// TIA Portal project "indexingStation" (V17)

(* hardware
DEVICE "SCALANCE X005"  SCALANCE X-Station
   slot 0: "Switch_1"  6GK5 005-0BA00-1AB2  V1.0
   slot 0: "SCALANCE X rack"  Rail
DEVICE "ET 200SP station_1"  ET 200SP-Station
   slot 0: "IO device_1"  IM 155-6 PN/2 HF  6ES7 155-6AU01-0CN0  V4.2
   slot 0: "Rack_0"  Rack  6ES5 710-8MAx1
   slot 1: "DI 8x24VDC HF_1"  DI 8x24VDC HF  6ES7 131-6BF00-0CA0  V2.0
      slot 1: "DI 8x24VDC HF_1"  DI 8x24VDC HF
   slot 2: "DI 8x24VDC HF_2"  DI 8x24VDC HF  6ES7 131-6BF00-0CA0  V2.0
      slot 1: "DI 8x24VDC HF_2"  DI 8x24VDC HF
   slot 3: "DI 8x24VDC HF_3"  DI 8x24VDC HF  6ES7 131-6BF00-0CA0  V2.0
      slot 1: "DI 8x24VDC HF_3"  DI 8x24VDC HF
   slot 4: "DQ 8x24VDC/0.5A HF_1"  DQ 8x24VDC/0.5A HF  6ES7 132-6BF00-0CA0  V2.0
      slot 1: "DQ 8x24VDC/0.5A HF_1"  DQ 8x24VDC/0.5A HF
   slot 5: "DQ 8x24VDC/0.5A HF_2"  DQ 8x24VDC/0.5A HF  6ES7 132-6BF00-0CA0  V2.0
      slot 1: "DQ 8x24VDC/0.5A HF_2"  DQ 8x24VDC/0.5A HF
   slot 6: "Server module_1"  Server module  6ES7 193-6PA00-0AA0  V1.1
      slot 1: "Server module_1"  Server module
   slot 127: "BA 2xRJ45"  BA 2xRJ45  6ES7 193-6AR00-0AA0  V0.0
      slot 1: "Port_1"  X1 P1 R  6ES7 193-6AR00-0AA0  V0.0
      slot 2: "Port_2"  X1 P2 R  6ES7 193-6AR00-0AA0  V0.0
DEVICE "S7-1200 station_1"  S7-1200 Station
   slot 0: "Rack_0"  S7-1200 Rack  Rack  V1.0
   slot 1: "PLC_1"  CPU 1214C DC/DC/DC  6ES7 214-1AG40-0XB0  V4.4
*)

// ===== PLC "PLC_1"  CPU 1214C DC/DC/DC =====

VAR_GLOBAL   // PLC tag table "Default tag table"
   "wrong orientation" AT %M10.0 : Bool;
   "Tag_1" AT %M202.1 : Bool;
   "end check" AT %M10.1 : Bool;
   "start correction" AT %M10.2 : Bool;
   "Tag_2" AT %M202.2 : Bool;
   "initiateGripper" AT %M10.3 : Bool;
   "initiateLifting" AT %M10.4 : Bool;
   "initiateRotation" AT %M10.5 : Bool;
   "initiateReturn" AT %M10.6 : Bool;
   "Tag_3" AT %M202.3 : Bool;
   "initiateOpenGripper" AT %M10.7 : Bool;
   "initiateNormalcy" AT %M11.0 : Bool;
   "Tag_4" AT %M202.4 : Bool;
   "initiateStepperMotor" AT %M11.1 : Bool;
   "prepForTransfer" AT %M11.2 : Bool;
   "initiateRetractionAfterTransfer" AT %M11.3 : Bool;
   "Clock_Byte" AT %MB50 : Byte;
   "Clock_10Hz" AT %M50.0 : Bool;
   "Clock_5Hz" AT %M50.1 : Bool;
   "Clock_2.5Hz" AT %M50.2 : Bool;
   "Clock_2Hz" AT %M50.3 : Bool;
   "Clock_1.25Hz" AT %M50.4 : Bool;
   "Clock_1Hz" AT %M50.5 : Bool;
   "Clock_0.625Hz" AT %M50.6 : Bool;
   "Clock_0.5Hz" AT %M50.7 : Bool;
   "rotate for check" AT %M11.4 : Bool;
   "rotate 90 if correct" AT %M11.5 : Bool;
   "rotate 45 if correct" AT %M11.6 : Bool;
   "rotate45 if incorrect" AT %M11.7 : Bool;
   "rotate 90 after incorrect orientation" AT %M12.0 : Bool;
END_VAR

VAR_GLOBAL   // PLC tag table "OurInputsAndOutputs"
   "Auto switch" AT %I0.6 : Bool;
   "reset Switch" AT %I0.5 : Bool;
   "start button" AT %I2.3 : Bool;
   "stop button" AT %I2.4 : Bool;
   "emergency stop" AT %I2.5 : Bool;
   "output power on" AT %I2.6 : Bool;
   "input 1 from previous station" AT %I2.7 : Bool;
   "input 2 from previous station" AT %I3.0 : Bool;
   "input 1 from next station" AT %I3.1 : Bool;
   "input 2 from next station" AT %I3.2 : Bool;
   "transfer cylinder 4A retracted" AT %I3.3 : Bool;
   "transfer cylinder 4A extended" AT %I3.4 : Bool;
   "lift cylinder 1A retracted" AT %I3.5 : Bool;
   "lift cylinder 1A extended" AT %I3.6 : Bool;
   "port present(orientationposition)" AT %I3.7 : Bool;
   "rotation cylinder 2A retracted" AT %I4.0 : Bool;
   "rotation cylinder 2A extended" AT %I4.1 : Bool;
   "Spool upper port detected" AT %I4.2 : Bool;
   "indexing station in home position" AT %I4.3 : Bool;
   "stepper motor ready" AT %I4.4 : Bool;
   "part present(initial position)" AT %I4.5 : Bool;
   "automatic on(green)" AT %Q2.0 : Bool;
   "output 1 to previous station" AT %Q2.1 : Bool;
   "output 2 to previous station" AT %Q2.2 : Bool;
   "output 1 to next station" AT %Q2.3 : Bool;
   "output 2 to next station" AT %Q2.4 : Bool;
   "extend transfer cylinder 3A" AT %Q2.5 : Bool;
   "extend lift cylinder" AT %Q2.6 : Bool;
   "retract lift cylinder" AT %Q2.7 : Bool;
   "stepper motor M1 go 45" AT %Q3.2 : Bool;
   "stepper motor M1 go 90" AT %Q3.3 : Bool;
   "release gripper 3A" AT %Q3.4 : Bool;
   "close gripper 3A" AT %Q3.5 : Bool;
   "extend rotation cylinder" AT %Q3.6 : Bool;
   "retract rotatioin cylinder" AT %Q3.7 : Bool;
END_VAR

// folder: System blocks/Program resources

DATA_BLOCK "timer 1"   // DB1
{ S7_Optimized_Access := 'TRUE' }
AUTHOR : Simatic
FAMILY : IEC
NAME : IEC_TMR
VERSION : 1.0
// stored: InstanceOfName IEC_TIMER
"IEC_TIMER"
BEGIN
END_DATA_BLOCK

DATA_BLOCK "timer 2"   // DB3
{ S7_Optimized_Access := 'TRUE' }
AUTHOR : Simatic
FAMILY : IEC
NAME : IEC_TMR
VERSION : 1.0
// stored: InstanceOfName IEC_TIMER
"IEC_TIMER"
BEGIN
END_DATA_BLOCK

DATA_BLOCK "timer 3"   // DB4
{ S7_Optimized_Access := 'TRUE' }
AUTHOR : Simatic
FAMILY : IEC
NAME : IEC_TMR
VERSION : 1.0
// stored: InstanceOfName IEC_TIMER
"IEC_TIMER"
BEGIN
END_DATA_BLOCK

DATA_BLOCK "timer 4"   // DB5
{ S7_Optimized_Access := 'TRUE' }
AUTHOR : Simatic
FAMILY : IEC
NAME : IEC_TMR
VERSION : 1.0
// stored: InstanceOfName IEC_TIMER
"IEC_TIMER"
BEGIN
END_DATA_BLOCK

// folder: (top level)

FUNCTION "correct orientation" : Void   // FC1, LAD
{ S7_Optimized_Access := 'TRUE' }
VERSION : 0.1
BEGIN

REGION Network 1: moving the stepper motor by 135 degrees
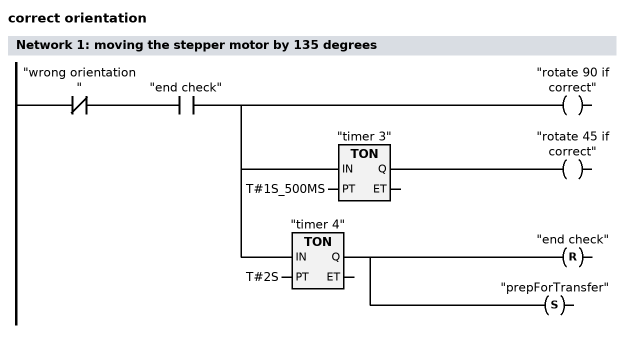
   "rotate 90 if correct" := NOT "wrong orientation" AND "end check";
   "timer 3".TON(IN := "rotate 90 if correct", PT := T#1S_500MS);
   "rotate 45 if correct" := "timer 3".Q;
   "timer 4".TON(IN := "rotate 90 if correct", PT := T#2S);
   IF "timer 4".Q THEN
       "end check" := FALSE;
       "prepForTransfer" := TRUE;
   END_IF;
END_REGION
END_FUNCTION

FUNCTION "incorrect orientation" : Void   // FC2, LAD
{ S7_Optimized_Access := 'TRUE' }
VERSION : 0.1
   VAR_TEMP   // added for the SCL form of the ladder/FBD networks
      _w1 : Bool;
   END_VAR
BEGIN

REGION Network 1: Launching of the correction procedure
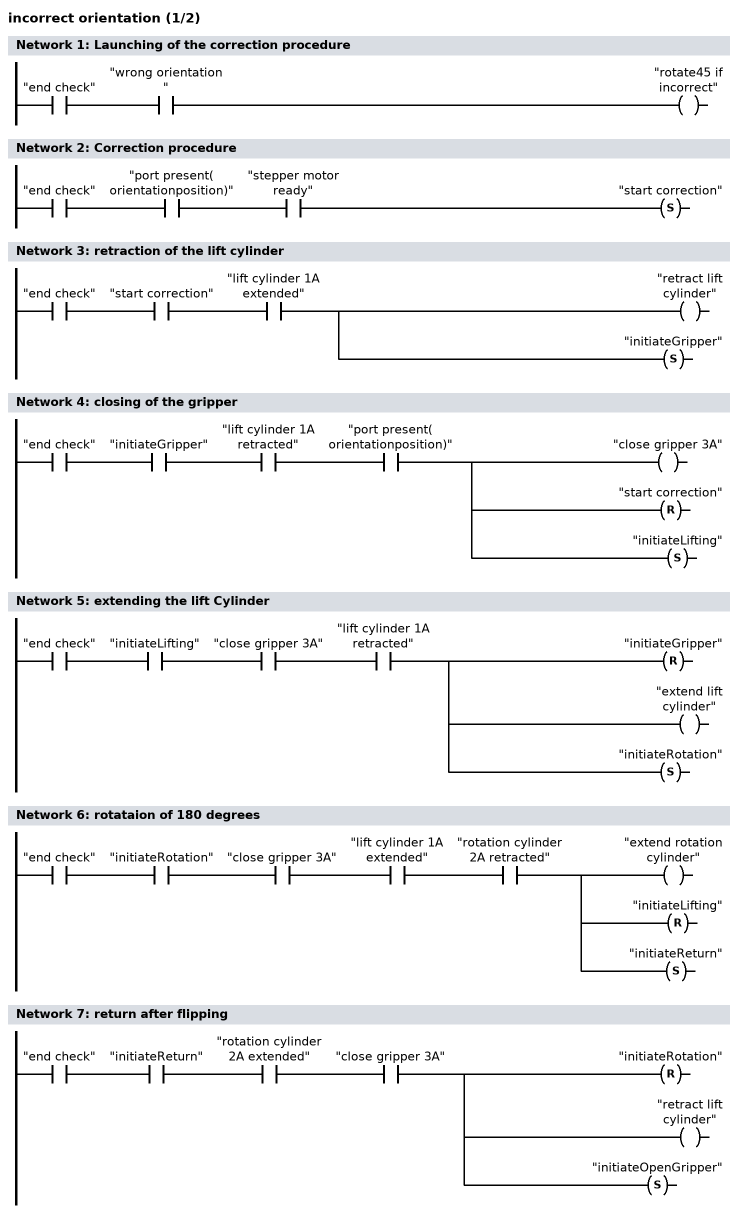
   RUNG wire#powerrail
      Contact( "end check" )
      Contact( "wrong orientation" )
      Coil( "rotate45 if incorrect" )
   END_RUNG
   // the same network as SCL:
   "rotate45 if incorrect" := "end check" AND "wrong orientation";
END_REGION

REGION Network 2: Correction procedure
   RUNG wire#powerrail
      Contact( "end check" )
      Contact( "port present(orientationposition)" )
      Contact( "stepper motor ready" )
      S_Coil( "start correction" )
   END_RUNG
   // the same network as SCL:
   IF "end check" AND "port present(orientationposition)" AND "stepper motor ready" THEN
       "start correction" := TRUE;
   END_IF;
END_REGION

REGION Network 3: retraction of the lift cylinder
   RUNG wire#powerrail
      Contact( "end check" )
      Contact( "start correction" )
      Contact( "lift cylinder 1A extended" )
      wire#w1
      Coil( "retract lift cylinder" )
   END_RUNG
   RUNG wire#w1
      S_Coil( "initiateGripper" )
   END_RUNG
   // the same network as SCL:
   "retract lift cylinder" := "end check" AND "start correction" AND "lift cylinder 1A extended";
   IF "retract lift cylinder" THEN "initiateGripper" := TRUE; END_IF;
END_REGION

REGION Network 4: closing of the gripper
   RUNG wire#powerrail
      Contact( "end check" )
      Contact( "initiateGripper" )
      Contact( "lift cylinder 1A retracted" )
      Contact( "port present(orientationposition)" )
      wire#w1
      Coil( "close gripper 3A" )
   END_RUNG
   RUNG wire#w1
      R_Coil( "start correction" )
   END_RUNG
   RUNG wire#w1
      S_Coil( "initiateLifting" )
   END_RUNG
   // the same network as SCL:
   "close gripper 3A" := "end check" AND "initiateGripper" AND "lift cylinder 1A retracted" AND "port present(orientationposition)";
   IF "close gripper 3A" THEN
       "start correction" := FALSE;
       "initiateLifting" := TRUE;
   END_IF;
END_REGION

REGION Network 5: extending the lift Cylinder
   RUNG wire#powerrail
      Contact( "end check" )
      Contact( "initiateLifting" )
      Contact( "close gripper 3A" )
      Contact( "lift cylinder 1A retracted" )
      wire#w1
      R_Coil( "initiateGripper" )
   END_RUNG
   RUNG wire#w1
      Coil( "extend lift cylinder" )
   END_RUNG
   RUNG wire#w1
      S_Coil( "initiateRotation" )
   END_RUNG
   // the same network as SCL:
   #_w1 := "end check" AND "initiateLifting" AND "close gripper 3A" AND "lift cylinder 1A retracted";
   IF #_w1 THEN "initiateGripper" := FALSE; END_IF;
   "extend lift cylinder" := #_w1;
   IF #_w1 THEN "initiateRotation" := TRUE; END_IF;
END_REGION

REGION Network 6: rotataion of 180 degrees
   RUNG wire#powerrail
      Contact( "end check" )
      Contact( "initiateRotation" )
      Contact( "close gripper 3A" )
      Contact( "lift cylinder 1A extended" )
      Contact( "rotation cylinder 2A retracted" )
      wire#w1
      Coil( "extend rotation cylinder" )
   END_RUNG
   RUNG wire#w1
      R_Coil( "initiateLifting" )
   END_RUNG
   RUNG wire#w1
      S_Coil( "initiateReturn" )
   END_RUNG
   // the same network as SCL:
   "extend rotation cylinder" := "end check" AND "initiateRotation" AND "close gripper 3A" AND "lift cylinder 1A extended" AND "rotation cylinder 2A retracted";
   IF "extend rotation cylinder" THEN
       "initiateLifting" := FALSE;
       "initiateReturn" := TRUE;
   END_IF;
END_REGION

REGION Network 7: return after flipping
   RUNG wire#powerrail
      Contact( "end check" )
      Contact( "initiateReturn" )
      Contact( "rotation cylinder 2A extended" )
      Contact( "close gripper 3A" )
      wire#w1
      R_Coil( "initiateRotation" )
   END_RUNG
   RUNG wire#w1
      Coil( "retract lift cylinder" )
   END_RUNG
   RUNG wire#w1
      S_Coil( "initiateOpenGripper" )
   END_RUNG
   // the same network as SCL:
   #_w1 := "end check" AND "initiateReturn" AND "rotation cylinder 2A extended" AND "close gripper 3A";
   IF #_w1 THEN "initiateRotation" := FALSE; END_IF;
   "retract lift cylinder" := #_w1;
   IF #_w1 THEN "initiateOpenGripper" := TRUE; END_IF;
END_REGION

REGION Network 8: releasing gripper
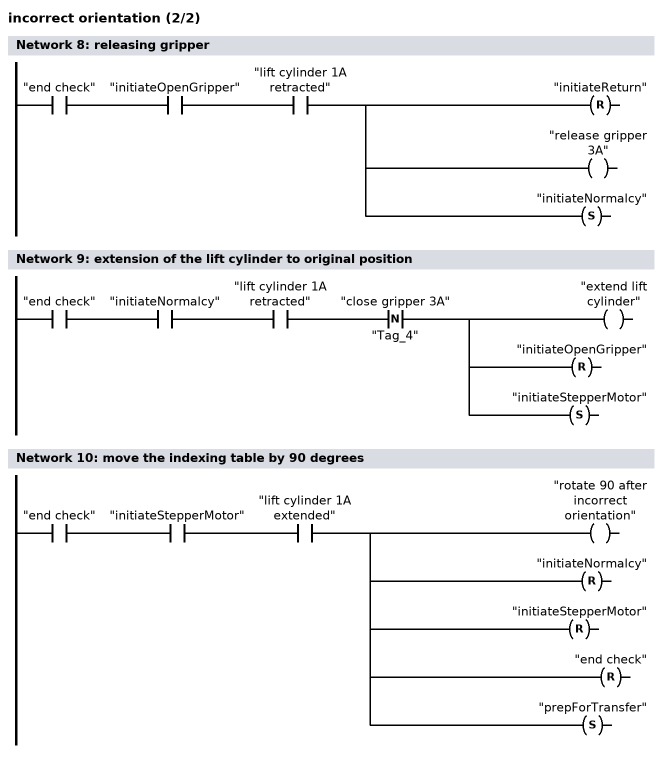
   RUNG wire#powerrail
      Contact( "end check" )
      Contact( "initiateOpenGripper" )
      Contact( "lift cylinder 1A retracted" )
      wire#w1
      R_Coil( "initiateReturn" )
   END_RUNG
   RUNG wire#w1
      Coil( "release gripper 3A" )
   END_RUNG
   RUNG wire#w1
      S_Coil( "initiateNormalcy" )
   END_RUNG
   // the same network as SCL:
   #_w1 := "end check" AND "initiateOpenGripper" AND "lift cylinder 1A retracted";
   IF #_w1 THEN "initiateReturn" := FALSE; END_IF;
   "release gripper 3A" := #_w1;
   IF #_w1 THEN "initiateNormalcy" := TRUE; END_IF;
END_REGION

REGION Network 9: extension of the lift cylinder to original position
   RUNG wire#powerrail
      Contact( "end check" )
      Contact( "initiateNormalcy" )
      Contact( "lift cylinder 1A retracted" )
      N_Contact(operand := "close gripper 3A", bit := "Tag_4")
      wire#w1
      Coil( "extend lift cylinder" )
   END_RUNG
   RUNG wire#w1
      R_Coil( "initiateOpenGripper" )
   END_RUNG
   RUNG wire#w1
      S_Coil( "initiateStepperMotor" )
   END_RUNG
   // the same network as SCL:
   #_w1 := "end check" AND "initiateNormalcy" AND "lift cylinder 1A retracted" AND NOT "close gripper 3A" AND "Tag_4";   // falling edge of "close gripper 3A"
   "Tag_4" := "close gripper 3A";
   "extend lift cylinder" := #_w1;
   IF #_w1 THEN
       "initiateOpenGripper" := FALSE;
       "initiateStepperMotor" := TRUE;
   END_IF;
END_REGION

REGION Network 10: move the indexing table by 90 degrees
   RUNG wire#powerrail
      Contact( "end check" )
      Contact( "initiateStepperMotor" )
      Contact( "lift cylinder 1A extended" )
      wire#w1
      Coil( "rotate 90 after incorrect orientation" )
   END_RUNG
   RUNG wire#w1
      R_Coil( "initiateNormalcy" )
   END_RUNG
   RUNG wire#w1
      R_Coil( "initiateStepperMotor" )
   END_RUNG
   RUNG wire#w1
      R_Coil( "end check" )
   END_RUNG
   RUNG wire#w1
      S_Coil( "prepForTransfer" )
   END_RUNG
   // the same network as SCL:
   "rotate 90 after incorrect orientation" := "end check" AND "initiateStepperMotor" AND "lift cylinder 1A extended";
   IF "rotate 90 after incorrect orientation" THEN
       "initiateNormalcy" := FALSE;
       "initiateStepperMotor" := FALSE;
       "end check" := FALSE;
       "prepForTransfer" := TRUE;
   END_IF;
END_REGION
END_FUNCTION

FUNCTION "Block_1" : Void   // FC3, LAD
{ S7_Optimized_Access := 'TRUE' }
VERSION : 0.1
BEGIN

REGION Network 1
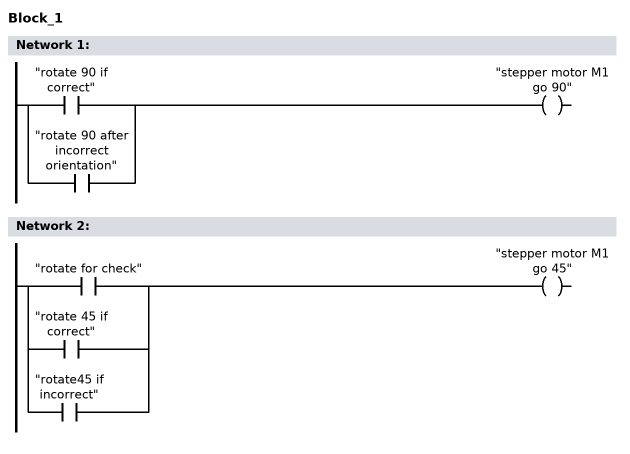
   RUNG wire#powerrail
      Contact( "rotate 90 if correct" )
      wire#w1
      Coil( "stepper motor M1 go 90" )
   END_RUNG
   RUNG wire#powerrail
      Contact( "rotate 90 after incorrect orientation" )
   END_RUNG wire#w1
   // the same network as SCL:
   "stepper motor M1 go 90" := "rotate 90 if correct" OR "rotate 90 after incorrect orientation";
END_REGION

REGION Network 2
   RUNG wire#powerrail
      Contact( "rotate for check" )
      wire#w1
      Coil( "stepper motor M1 go 45" )
   END_RUNG
   RUNG wire#powerrail
      Contact( "rotate 45 if correct" )
   END_RUNG wire#w1
   RUNG wire#powerrail
      Contact( "rotate45 if incorrect" )
   END_RUNG wire#w1
   // the same network as SCL:
   "stepper motor M1 go 45" := "rotate for check" OR "rotate 45 if correct" OR "rotate45 if incorrect";
END_REGION
END_FUNCTION

ORGANIZATION_BLOCK "Main"   // OB1, LAD, ProgramCycle
TITLE = "Main Program Sweep (Cycle)"
{ S7_Optimized_Access := 'TRUE' }
VERSION : 0.1
   VAR_INPUT
      Initial_Call : Bool;   // Initial call of this OB
      Remanence : Bool;   // =True, if remanent data are available
   END_VAR
   VAR_TEMP   // added for the SCL form of the ladder/FBD networks
      _w1 : Bool;
   END_VAR
BEGIN

REGION Network 1: Stepper motor go 45
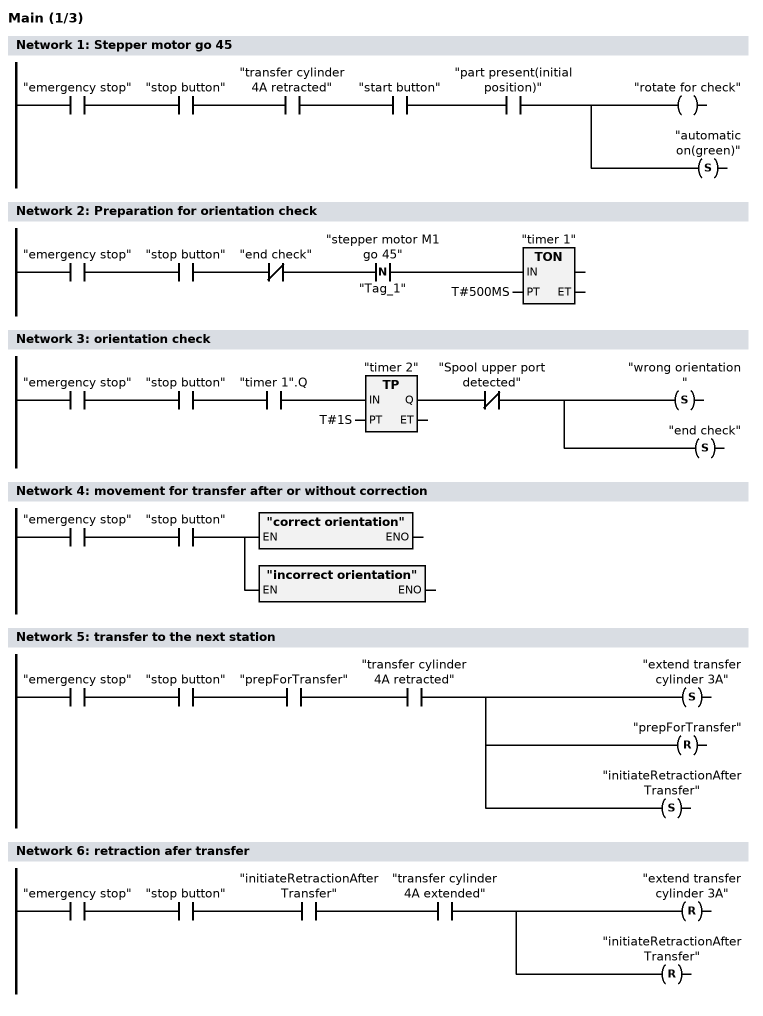
   RUNG wire#powerrail
      Contact( "emergency stop" )
      Contact( "stop button" )
      Contact( "transfer cylinder 4A retracted" )
      Contact( "start button" )
      Contact( "part present(initial position)" )
      wire#w1
      Coil( "rotate for check" )
   END_RUNG
   RUNG wire#w1
      S_Coil( "automatic on(green)" )
   END_RUNG
   // the same network as SCL:
   "rotate for check" := "emergency stop" AND "stop button" AND "transfer cylinder 4A retracted" AND "start button" AND "part present(initial position)";
   IF "rotate for check" THEN "automatic on(green)" := TRUE; END_IF;
END_REGION

REGION Network 2: Preparation for orientation check
   #_w1 := "emergency stop" AND "stop button" AND NOT "end check" AND NOT "stepper motor M1 go 45" AND "Tag_1";   // falling edge of "stepper motor M1 go 45"
   "Tag_1" := "stepper motor M1 go 45";
   "timer 1".TON(IN := #_w1, PT := T#500MS);
END_REGION

REGION Network 3: orientation check
   "timer 2".TP(IN := "emergency stop" AND "stop button" AND "timer 1".Q, PT := T#1S);
   IF "timer 2".Q AND NOT "Spool upper port detected" THEN
       "wrong orientation" := TRUE;
       "end check" := TRUE;
   END_IF;
END_REGION

REGION Network 4: movement for transfer after or without correction
   RUNG wire#powerrail
      Contact( "emergency stop" )
      Contact( "stop button" )
      wire#w1
      "correct orientation"()
   END_RUNG
   RUNG wire#w1
      "incorrect orientation"()
   END_RUNG
   // the same network as SCL:
   #_w1 := "emergency stop" AND "stop button";
   IF #_w1 THEN
       "correct orientation"();
       "incorrect orientation"();
   END_IF;
END_REGION

REGION Network 5: transfer to the next station
   RUNG wire#powerrail
      Contact( "emergency stop" )
      Contact( "stop button" )
      Contact( "prepForTransfer" )
      Contact( "transfer cylinder 4A retracted" )
      wire#w1
      S_Coil( "extend transfer cylinder 3A" )
   END_RUNG
   RUNG wire#w1
      R_Coil( "prepForTransfer" )
   END_RUNG
   RUNG wire#w1
      S_Coil( "initiateRetractionAfterTransfer" )
   END_RUNG
   // the same network as SCL:
   IF "emergency stop" AND "stop button" AND "prepForTransfer" AND "transfer cylinder 4A retracted" THEN
       "extend transfer cylinder 3A" := TRUE;
   END_IF;
   #_w1 := "emergency stop" AND "stop button" AND "prepForTransfer" AND "transfer cylinder 4A retracted";
   IF #_w1 THEN
       "prepForTransfer" := FALSE;
       "initiateRetractionAfterTransfer" := TRUE;
   END_IF;
END_REGION

REGION Network 6: retraction afer transfer
   RUNG wire#powerrail
      Contact( "emergency stop" )
      Contact( "stop button" )
      Contact( "initiateRetractionAfterTransfer" )
      Contact( "transfer cylinder 4A extended" )
      wire#w1
      R_Coil( "extend transfer cylinder 3A" )
   END_RUNG
   RUNG wire#w1
      R_Coil( "initiateRetractionAfterTransfer" )
   END_RUNG
   // the same network as SCL:
   IF "emergency stop" AND "stop button" AND "initiateRetractionAfterTransfer" AND "transfer cylinder 4A extended" THEN
       "extend transfer cylinder 3A" := FALSE;
       "initiateRetractionAfterTransfer" := FALSE;
   END_IF;
END_REGION

REGION Network 7: reset action
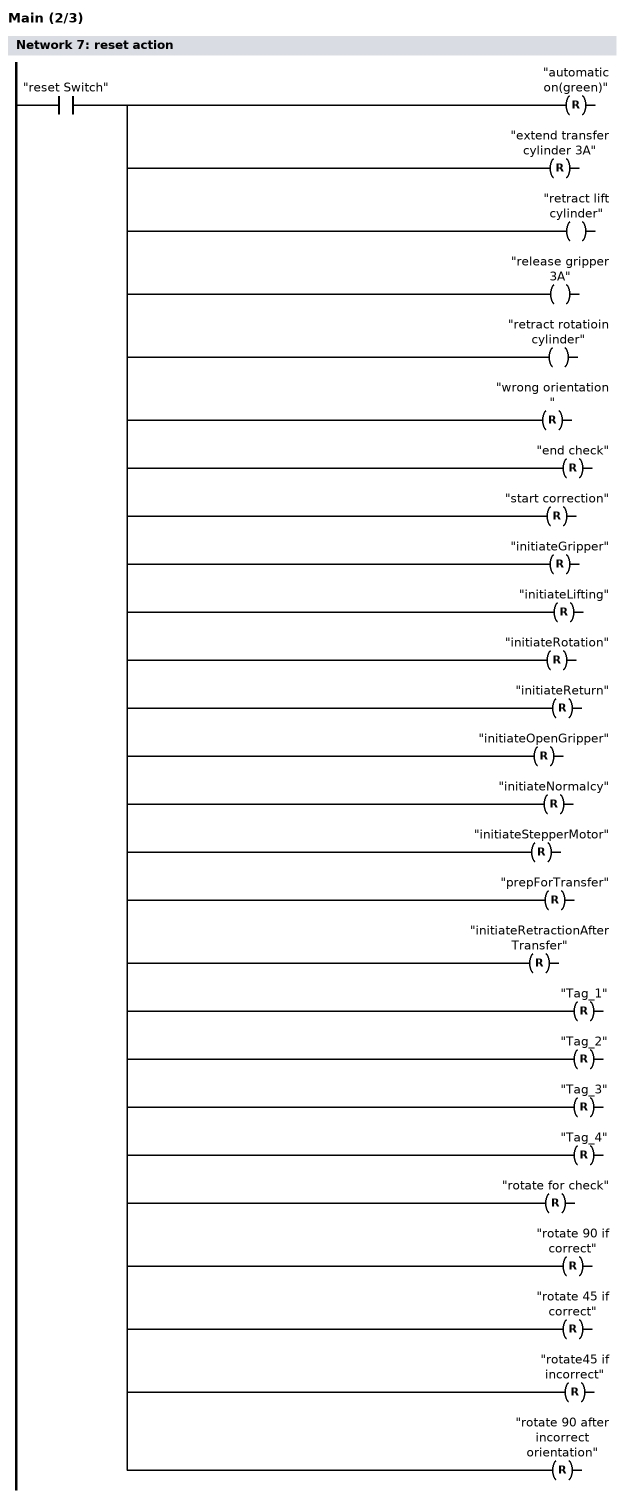
   RUNG wire#powerrail
      Contact( "reset Switch" )
      wire#w1
      R_Coil( "automatic on(green)" )
   END_RUNG
   RUNG wire#w1
      R_Coil( "extend transfer cylinder 3A" )
   END_RUNG
   RUNG wire#w1
      Coil( "retract lift cylinder" )
   END_RUNG
   RUNG wire#w1
      Coil( "release gripper 3A" )
   END_RUNG
   RUNG wire#w1
      Coil( "retract rotatioin cylinder" )
   END_RUNG
   RUNG wire#w1
      R_Coil( "wrong orientation" )
   END_RUNG
   RUNG wire#w1
      R_Coil( "end check" )
   END_RUNG
   RUNG wire#w1
      R_Coil( "start correction" )
   END_RUNG
   RUNG wire#w1
      R_Coil( "initiateGripper" )
   END_RUNG
   RUNG wire#w1
      R_Coil( "initiateLifting" )
   END_RUNG
   RUNG wire#w1
      R_Coil( "initiateRotation" )
   END_RUNG
   RUNG wire#w1
      R_Coil( "initiateReturn" )
   END_RUNG
   RUNG wire#w1
      R_Coil( "initiateOpenGripper" )
   END_RUNG
   RUNG wire#w1
      R_Coil( "initiateNormalcy" )
   END_RUNG
   RUNG wire#w1
      R_Coil( "initiateStepperMotor" )
   END_RUNG
   RUNG wire#w1
      R_Coil( "prepForTransfer" )
   END_RUNG
   RUNG wire#w1
      R_Coil( "initiateRetractionAfterTransfer" )
   END_RUNG
   RUNG wire#w1
      R_Coil( "Tag_1" )
   END_RUNG
   RUNG wire#w1
      R_Coil( "Tag_2" )
   END_RUNG
   RUNG wire#w1
      R_Coil( "Tag_3" )
   END_RUNG
   RUNG wire#w1
      R_Coil( "Tag_4" )
   END_RUNG
   RUNG wire#w1
      R_Coil( "rotate for check" )
   END_RUNG
   RUNG wire#w1
      R_Coil( "rotate 90 if correct" )
   END_RUNG
   RUNG wire#w1
      R_Coil( "rotate 45 if correct" )
   END_RUNG
   RUNG wire#w1
      R_Coil( "rotate45 if incorrect" )
   END_RUNG
   RUNG wire#w1
      R_Coil( "rotate 90 after incorrect orientation" )
   END_RUNG
   // the same network as SCL:
   IF "reset Switch" THEN
       "automatic on(green)" := FALSE;
       "extend transfer cylinder 3A" := FALSE;
   END_IF;
   "retract lift cylinder" := "reset Switch";
   "release gripper 3A" := "reset Switch";
   "retract rotatioin cylinder" := "reset Switch";
   IF "reset Switch" THEN
       "wrong orientation" := FALSE;
       "end check" := FALSE;
       "start correction" := FALSE;
       "initiateGripper" := FALSE;
       "initiateLifting" := FALSE;
       "initiateRotation" := FALSE;
       "initiateReturn" := FALSE;
       "initiateOpenGripper" := FALSE;
       "initiateNormalcy" := FALSE;
       "initiateStepperMotor" := FALSE;
       "prepForTransfer" := FALSE;
       "initiateRetractionAfterTransfer" := FALSE;
       "Tag_1" := FALSE;
       "Tag_2" := FALSE;
       "Tag_3" := FALSE;
       "Tag_4" := FALSE;
       "rotate for check" := FALSE;
       "rotate 90 if correct" := FALSE;
       "rotate 45 if correct" := FALSE;
       "rotate45 if incorrect" := FALSE;
       "rotate 90 after incorrect orientation" := FALSE;
   END_IF;
END_REGION

REGION Network 8
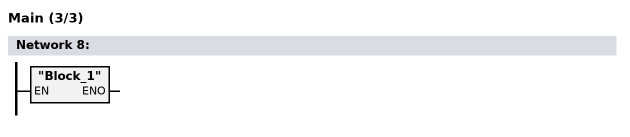
   RUNG wire#powerrail
      "Block_1"()
   END_RUNG
   // the same network as SCL:
   "Block_1"();
END_REGION
END_ORGANIZATION_BLOCK